(* IEC 61131-3 sources: MotionTestBenchMaster/Logical/00_AID/Libraries/System_Libraries/AsICMP, 3 files *)

(* ---- AsICMP.typ ---- *)
(********************************************************************
 * COPYRIGHT -- Bernecker + Rainer
 ********************************************************************
 * Library: AsICMP
 * File: AsICMP.typ
 * Author: B+R
 ********************************************************************
 * Data types of library AsICMP
 ********************************************************************)

TYPE

END_TYPE

(* ---- AsICMP.fun ---- *)
(********************************************************************
 * COPYRIGHT -- Bernecker + Rainer
 ********************************************************************
 * Library: AsIcmp
 * File: AsIcmp.fun
 * Author: B+R
 ********************************************************************
 * Functions and function blocks of library AsIcmp
 ********************************************************************)

{REDUND_CONTEXT} {REDUND_UNREPLICABLE} FUNCTION_BLOCK IcmpPing					(*pings a station; asynchronous execution*)
	VAR_INPUT
		enable			: BOOL;			(*enables execution*)
		pHost			: UDINT;		(*pointer to the IP address or name of the station that should be pinged*)
		timeout			: UINT;			(*response timeout*)
	END_VAR

	VAR_OUTPUT
		status			: UINT;			(*execution status: ERR_OK, ERR_FUB_ENABLE_FALSE, ERR_FUB_BUSY, 0xXXXX = see help*)
	END_VAR

	VAR
        i_state			: UINT;			(*internal variable*)
		i_result		: UINT;			(*internal variable*)
        i_tmp			: UDINT;		(*internal variable*)
	END_VAR
END_FUNCTION_BLOCK

(* ---- AsICMP.var ---- *)
(********************************************************************
 * COPYRIGHT -- Bernecker + Rainer
 ********************************************************************
 * Library: AsIcmp
 * File: AsIcmp.var
 * Author: B+R
 ********************************************************************
 * Local variables of library AsIcmp
 ********************************************************************)

VAR CONSTANT
	icmpERR_NO_RESPONSE					: UINT := 32750;	(*no ping response*)
	icmpERR_PARAMETER					: UINT := 32751;	(*invalid parameter, check parameter*)
	icmpERR_SOCKET_CREATE				: UINT := 32752;	(*create socket failed*)
	icmpERR_UNREACHABLE					: UINT := 32753;	(*host unreachable*)
	icmpERR_SYSTEM						: UINT := 32799;	(*system error*)
END_VAR
